# B&R Automation Studio project Panasonic_LinkaPowerCP2_A2021055 (part 11)

```iecst
			IF NOT SC_P1_StoperSrobovania.Switch1 THEN
				P1_Skrutk_5H_PravaM5_Vysunutie:= STRING_TO_REAL(Reports.Skrutkovacky.VyskaSkrutkovania.P1_PravaSkrutkaM5);
				IF (P1_Skrutk_5H_PravaM5_Vysunutie <= P1_RemPremenne.P1_Srob5H_PravaM5_Vysunutie_HI) AND (P1_Skrutk_5H_PravaM5_Vysunutie >= P1_RemPremenne.P1_Srob5H_PravaM5_Vysunutie_LO) THEN
					VysunutieSkrutkovacky_OK:= TRUE;
				ELSE
					VysunutieSkrutkovacky_OK:= FALSE;
				END_IF
				SC_P1_StoperSrobovania.Switch1:= TRUE;
			END_IF

			IF P1_Srobovanie.STAV.Vysledok_Srobovania = 'OK' THEN
				IF VysunutieSkrutkovacky_OK THEN
					Reports.Skrutkovacky.VyslednyReport.P1_PravaSkrutkaM5:= 'PASS';
					SC_P1_StoperSrobovania.ResetStep:= TRUE;
					SC_P1_StoperSrobovania.Step:= 390;
				ELSE
					Reports.Skrutkovacky.VyslednyReport.P1_PravaSkrutkaM5:= 'FAIL';
					IF P1_Srobov_M5_Result_OFF THEN
						SC_P1_StoperSrobovania.ResetStep:= TRUE;
						SC_P1_StoperSrobovania.Step:= 390;
					ELSE
						Paletka[i].PAR.StavPowerCP:= 'FAIL';
						Paletka[i].STAV.StavPaletky:= 'NG';
						SC_P1_StoperSrobovania.ResetStep:= TRUE;
						SC_P1_StoperSrobovania.Step:= 500;
					END_IF
				END_IF
			ELSIF P1_Srobovanie.STAV.Vysledok_Srobovania = 'NG' THEN
				Reports.Skrutkovacky.VyslednyReport.P1_PravaSkrutkaM5:= 'FAIL';
				IF P1_Srobov_M5_Result_OFF THEN
					SC_P1_StoperSrobovania.ResetStep:= TRUE;
					SC_P1_StoperSrobovania.Step:= 390;
				ELSE
					Paletka[i].PAR.StavPowerCP:= 'FAIL';
					Paletka[i].STAV.StavPaletky:= 'NG';
					SC_P1_StoperSrobovania.ResetStep:= TRUE;
					SC_P1_StoperSrobovania.Step:= 500;
				END_IF
			END_IF

		390:
			SC_P1_StoperSrobovania.StepName:='390 - Automaticky Rezim - model 5H odobratie skrutky M5';
			SC_P1_StoperSrobovania.IdleTime.PT:= T#200ms;
			SC_P1_StoperSrobovania.AlarmTime.PT:= T#5s;

			IF NOT SC_P1_StoperSrobovania.Switch1  THEN
				P1_Srobovanie.COM_IN.OdoberSkrutku_M5:= TRUE;
				SC_P1_StoperSrobovania.Switch1:= TRUE;
			END_IF

			IF P1_Srobovanie.STAV.ManipulatorNadPodavacmi THEN
				P1_Srobovanie.COM_IN.OdoberSkrutku_M5:= FALSE;
				SC_P1_StoperSrobovania.ResetStep:= TRUE;
				SC_P1_StoperSrobovania.Step:= 391;
			END_IF

		391:
			SC_P1_StoperSrobovania.StepName:='391 - Automaticky Rezim - cakam na zrusenie signalu presun manipulatora ukonceny';
			SC_P1_StoperSrobovania.IdleTime.PT:= T#200ms;
			SC_P1_StoperSrobovania.AlarmTime.PT:= T#5s;

			IF NOT P1_Robot.COM_IN.Stav_RobotPoziciaCakania THEN
				SC_P1_StoperSrobovania.ResetStep:= TRUE;
				SC_P1_StoperSrobovania.Step:= 392;
			END_IF

		392:
			SC_P1_StoperSrobovania.StepName:='392 - Automaticky Rezim - model 5H vystavenie signalu pre robota chod do cakacej pozicie';
			SC_P1_StoperSrobovania.IdleTime.PT:= T#200ms;
			SC_P1_StoperSrobovania.AlarmTime.PT:= T#5s;

			P1_Robot.COM_OUT.ManipSrobovania_BezpecnaPozicia:= TRUE;

			IF NOT SC_P1_StoperSrobovania.Switch1 THEN
				P1_Robot.COM_OUT.Presun_CakaciaPozicia:= TRUE;
				SC_P1_StoperSrobovania.Switch1:= TRUE;
			END_IF

			IF P1_Robot.COM_IN.Stav_RobotPoziciaCakania AND NOT P1_Srobovanie.COM_OUT.Stav_SkrutkovanieUkoncene THEN
				P1_Robot.COM_OUT.Presun_CakaciaPozicia:= FALSE;
				CAM6.STAV.Results_READY:= FALSE;
				CAM6.STAV.OldRunCounter:= CAM6.STAV.RunCounter;
				SC_P1_StoperSrobovania.ResetStep:= TRUE;
				SC_P1_StoperSrobovania.Step:= 395;
			END_IF

		395:
			SC_P1_StoperSrobovania.StepName:='395 - Inicializacia - model 5H kamerova kontrola paletky CAM6';//CAM 6//
			SC_P1_StoperSrobovania.IdleTime.PT:= T#5s;
			SC_P1_StoperSrobovania.AlarmTime.PT:= T#5s;

			IF NOT SC_P1_StoperSrobovania.Switch1 AND CAM6.STAV.Command_READY THEN
				CAM6.CMD.Triger:= TRUE;
				SC_P1_StoperSrobovania.IdleTime.IN:= TRUE;
				SC_P1_StoperSrobovania.Switch1:= TRUE;
			END_IF

			IF CAM6.STAV.Results_READY AND CAM6.STAV.Command_AKCEPTOVANY AND CAM6.STAV.OldRunCounter <> CAM6.STAV.RunCounter THEN
				PocetTrigrovKamery:= 0;
				CAM6.STAV.Results_READY:= FALSE;
				CAM6.STAV.OldRunCounter:= CAM6.STAV.RunCounter;
				SC_P1_StoperSrobovania.ResetStep:= TRUE;
				SC_P1_StoperSrobovania.Step:= 398;
			ELSIF SC_P1_StoperSrobovania.IdleTime.Q AND PocetTrigrovKamery < 5 THEN
				PocetTrigrovKamery:= PocetTrigrovKamery + 1;
				CAM6.STAV.Results_READY:= FALSE;
				CAM6.STAV.OldRunCounter:= CAM6.STAV.RunCounter;
				CAM6.CMD.Triger:= FALSE;
				SC_P1_StoperSrobovania.ResetStep:= TRUE;
				SC_P1_StoperSrobovania.Step:= 397;
			ELSIF SC_P1_StoperSrobovania.IdleTime.Q AND PocetTrigrovKamery >= 5 THEN
				P1_Alarmy[168]:= TRUE;
				P1_Pracovisko.STAV.Porucha_ST2:= TRUE;
			END_IF

		397:
			SC_P1_StoperSrobovania.StepName:='397 - Automaticky Rezim - cakam na opatovny triger kamery CAM6';
			SC_P1_StoperSrobovania.IdleTime.PT:= T#1s;
			SC_P1_StoperSrobovania.AlarmTime.PT:= T#5s;

			SC_P1_StoperSrobovania.IdleTime.IN:= TRUE;

			IF SC_P1_StoperSrobovania.IdleTime.Q THEN
				SC_P1_StoperSrobovania.ResetStep:= TRUE;
				SC_P1_StoperSrobovania.Step:= 395;
			END_IF

		398:
			SC_P1_StoperSrobovania.StepName:='398 - Automaticky Rezim - model 5H kontrola vysledku kamery';
			SC_P1_StoperSrobovania.IdleTime.PT:= T#200ms;
			SC_P1_StoperSrobovania.AlarmTime.PT:= T#5s;
			SC_P1_StoperSrobovania.IdleTime.IN:= TRUE;

			IF Linka.P1_Kamery_OFF THEN
				CAM6.CMD.Triger:= FALSE;
				CAM6.PAR.ResultFotky:= 'PASS';
				SC_P1_StoperSrobovania.ResetStep:= TRUE;
				SC_P1_StoperSrobovania.Step:= 403;
			ELSIF NOT CAM6.STAV.BUSY THEN
				CAM6.CMD.Triger:= FALSE;
				IF NOT CAM6.RESULT.Paletka.Pritom_SpodnychBusbarov_5H AND
					CAM6.RESULT.PowerCP.Pritom_LavejSkrutkyK30 AND
					CAM6.RESULT.PowerCP.Pritom_PravejSkrutkyK30 THEN
					CAM6.PAR.ResultFotky:= 'PASS';
					SC_P1_StoperSrobovania.ResetStep:= TRUE;
					SC_P1_StoperSrobovania.Step:= 403;
				ELSE
					CAM6.PAR.ResultFotky:= 'FAIL';
					SC_P1_StoperSrobovania.ResetStep:= TRUE;
					SC_P1_StoperSrobovania.Step:= 403;
				END_IF
			END_IF

		403:
			SC_P1_StoperSrobovania.StepName:='403 - Automaticky Rezim - model 5H rozhodnutie podla kamerovej kontroly paletky';
			SC_P1_StoperSrobovania.IdleTime.PT:= T#200ms;
			SC_P1_StoperSrobovania.AlarmTime.PT:= T#5s;

			IF CAM6.PAR.ResultFotky = 'PASS' THEN
				Paletka[i].PAR.StavPowerCP:= 'PASS';
				SC_P1_StoperSrobovania.ResetStep:= TRUE;
				SC_P1_StoperSrobovania.Step:= 540;
			ELSIF CAM6.PAR.ResultFotky = 'FAIL' THEN
				P1_Vizu.ZobrazHL8_ST2:= TRUE;
				IF P1_Srobov_KAM_Result_OK THEN
					P1_Srobov_KAM_Result_OK:= FALSE;
					P1_Vizu.ZobrazHL8_ST2:= FALSE;
					Paletka[i].PAR.StavPowerCP:= 'PASS';
					CAM6.PAR.ResultFotky:= 'PASS';
					SC_P1_StoperSrobovania.ResetStep:= TRUE;
					SC_P1_StoperSrobovania.Step:= 540;
				ELSIF P1_Srobov_KAM_Result_NG THEN
					P1_Srobov_KAM_Result_NG:= FALSE;
					P1_Vizu.ZobrazHL8_ST2:= FALSE;
					Paletka[i].PAR.StavPowerCP:= 'FAIL';
					Paletka[i].STAV.StavPaletky:= 'NG';
					SC_P1_StoperSrobovania.ResetStep:= TRUE;
					SC_P1_StoperSrobovania.Step:= 540;
				END_IF
			END_IF

			//**************************Uvolnenie robota a vyfotenie paletky po zlom skrutkovaní*****************************************************//

		500:
			SC_P1_StoperSrobovania.StepName:='500 - Automaticky Rezim - presun manipulatora vzad';
			SC_P1_StoperSrobovania.IdleTime.PT:= T#200ms;
			SC_P1_StoperSrobovania.AlarmTime.PT:= T#5s;

			IF NOT SC_P1_StoperSrobovania.Switch1 THEN
				P1_Srobovanie.COM_IN.PresunManipulatora_VZAD:= TRUE;
				SC_P1_StoperSrobovania.Switch1:= TRUE;
			END_IF

			IF P1_Srobovanie.COM_OUT.Stav_PresunManipulUkonceny THEN
				P1_Srobovanie.COM_IN.PresunManipulatora_VZAD:= FALSE;
				SC_P1_StoperSrobovania.ResetStep:= TRUE;
				SC_P1_StoperSrobovania.Step:= 501;
			END_IF

		501:
			SC_P1_StoperSrobovania.StepName:='501 - Automaticky Rezim - cakam na zrusenie signalu presun manipulatora ukonceny';
			SC_P1_StoperSrobovania.IdleTime.PT:= T#200ms;
			SC_P1_StoperSrobovania.AlarmTime.PT:= T#5s;

			IF NOT P1_Srobovanie.COM_OUT.Stav_PresunManipulUkonceny THEN
				SC_P1_StoperSrobovania.ResetStep:= TRUE;
				SC_P1_StoperSrobovania.Step:= 503;
			END_IF

		503:
			SC_P1_StoperSrobovania.StepName:='503 - Automaticky Rezim - kontrola ci robot drzi foamy';
			SC_P1_StoperSrobovania.IdleTime.PT:= T#200ms;
			SC_P1_StoperSrobovania.AlarmTime.PT:= T#5s;

			IF Linka.PAR.ZvolenyModel = '4F' THEN
				IF P1_Robot.STAV.DrziFoamy_45F THEN
					P1_Robot.COM_OUT.PolozFoam4F_na_PowerCP:= TRUE;
					IF P1_Robot.COM_IN.Stav_Foam4F_Polozeny THEN
						P1_Robot.COM_OUT.PolozFoam4F_na_PowerCP:= FALSE;
						SC_P1_StoperSrobovania.ResetStep:= TRUE;
						SC_P1_StoperSrobovania.Step:= 505;
					END_IF
				ELSE
					SC_P1_StoperSrobovania.ResetStep:= TRUE;
					SC_P1_StoperSrobovania.Step:= 505;
				END_IF
			ELSIF Linka.PAR.ZvolenyModel = '5F' THEN
				IF P1_Robot.STAV.DrziFoamy_45F THEN
					P1_Robot.COM_OUT.PolozFoam5F_na_PowerCP:= TRUE;
					IF P1_Robot.COM_IN.Stav_Foam5F_Polozeny THEN
						P1_Robot.COM_OUT.PolozFoam5F_na_PowerCP:= FALSE;
						SC_P1_StoperSrobovania.ResetStep:= TRUE;
						SC_P1_StoperSrobovania.Step:= 505;
					END_IF
				ELSE
					SC_P1_StoperSrobovania.ResetStep:= TRUE;
					SC_P1_StoperSrobovania.Step:= 505;
				END_IF
			ELSIF Linka.PAR.ZvolenyModel = '5H' THEN
				SC_P1_StoperSrobovania.ResetStep:= TRUE;
				SC_P1_StoperSrobovania.Step:= 505;
			END_IF

		505:
			SC_P1_StoperSrobovania.StepName:='505 - Automaticky Rezim - kontrola ci robot drzi busbary';
			SC_P1_StoperSrobovania.IdleTime.PT:= T#200ms;
			SC_P1_StoperSrobovania.AlarmTime.PT:= T#5s;

			IF Linka.PAR.ZvolenyModel = '4F' THEN
				IF P1_Robot.STAV.DrziBusbar_45F THEN
					P1_Robot.COM_OUT.PolozSpodnyBusbar4F_na_PowerCP:= TRUE;
					IF P1_Robot.COM_IN.Stav_SpodnyBusbar4F_Polozeny THEN
						P1_Robot.COM_OUT.PolozSpodnyBusbar4F_na_PowerCP:= FALSE;
						SC_P1_StoperSrobovania.ResetStep:= TRUE;
						SC_P1_StoperSrobovania.Step:= 508;
					END_IF
				ELSE
					SC_P1_StoperSrobovania.ResetStep:= TRUE;
					SC_P1_StoperSrobovania.Step:= 508;
				END_IF
			ELSIF Linka.PAR.ZvolenyModel = '5F' THEN
				IF P1_Robot.STAV.DrziBusbar_45F THEN
					P1_Robot.COM_OUT.PolozSpodnyBusbar5F_na_PowerCP:= TRUE;
					IF P1_Robot.COM_IN.Stav_SpodnyBusbar5F_Polozeny THEN
						P1_Robot.COM_OUT.PolozSpodnyBusbar5F_na_PowerCP:= FALSE;
						SC_P1_StoperSrobovania.ResetStep:= TRUE;
						SC_P1_StoperSrobovania.Step:= 508;
					END_IF
				ELSE
					SC_P1_StoperSrobovania.ResetStep:= TRUE;
					SC_P1_StoperSrobovania.Step:= 508;
				END_IF
			ELSIF Linka.PAR.ZvolenyModel = '5H' THEN
				IF P1_Robot.STAV.DrziBusbar_5H THEN
					P1_Robot.COM_OUT.PolozSpodnyBusbar5H_na_PowerCP:= TRUE;
					IF P1_Robot.COM_IN.Stav_SpodnyBusbar5H_Polozeny THEN
						P1_Robot.COM_OUT.PolozSpodnyBusbar5H_na_PowerCP:= FALSE;
						SC_P1_StoperSrobovania.ResetStep:= TRUE;
						SC_P1_StoperSrobovania.Step:= 510;
					END_IF
				ELSE
					SC_P1_StoperSrobovania.ResetStep:= TRUE;
					SC_P1_StoperSrobovania.Step:= 510;
				END_IF
			END_IF

		508:
			SC_P1_StoperSrobovania.StepName:='508 - Automaticky Rezim - kontrola ci robot drzi DPS';
			SC_P1_StoperSrobovania.IdleTime.PT:= T#200ms;
			SC_P1_StoperSrobovania.AlarmTime.PT:= T#5s;

			IF Linka.PAR.ZvolenyModel = '4F' THEN
				IF P1_Robot.STAV.DrziDPS_45F THEN
					P1_Robot.COM_OUT.PolozDPS_4F_na_PowerCP:= TRUE;
					IF P1_Robot.COM_IN.Stav_DPS_4F_Polozeny THEN
						P1_Robot.COM_OUT.PolozDPS_4F_na_PowerCP:= FALSE;
						SC_P1_StoperSrobovania.ResetStep:= TRUE;
						SC_P1_StoperSrobovania.Step:= 510;
					END_IF
				ELSE
					SC_P1_StoperSrobovania.ResetStep:= TRUE;
					SC_P1_StoperSrobovania.Step:= 510;
				END_IF
			ELSIF Linka.PAR.ZvolenyModel = '5F' THEN
				IF P1_Robot.STAV.DrziDPS_45F THEN
					P1_Robot.COM_OUT.PolozDPS_5F_na_PowerCP:= TRUE;
					IF P1_Robot.COM_IN.Stav_DPS_5F_Polozeny THEN
						P1_Robot.COM_OUT.PolozDPS_5F_na_PowerCP:= FALSE;
						SC_P1_StoperSrobovania.ResetStep:= TRUE;
						SC_P1_StoperSrobovania.Step:= 510;
					END_IF
				ELSE
					SC_P1_StoperSrobovania.ResetStep:= TRUE;
					SC_P1_StoperSrobovania.Step:= 510;
				END_IF
			END_IF

		510:
			SC_P1_StoperSrobovania.StepName:='510 - Automaticky Rezim - vystavenie signalu pre robota chod do cakacej pozicie';
			SC_P1_StoperSrobovania.IdleTime.PT:= T#200ms;
			SC_P1_StoperSrobovania.AlarmTime.PT:= T#5s;

			P1_Robot.COM_OUT.ManipSrobovania_BezpecnaPozicia:= TRUE;

			IF NOT SC_P1_StoperSrobovania.Switch1 THEN
				P1_Robot.COM_OUT.Presun_CakaciaPozicia:= TRUE;
				SC_P1_StoperSrobovania.Switch1:= TRUE;
			END_IF

			IF P1_Robot.COM_IN.Stav_RobotPoziciaCakania THEN
				P1_Robot.COM_OUT.Presun_CakaciaPozicia:= FALSE;
				CAM6.STAV.Results_READY:= FALSE;
				CAM6.STAV.OldRunCounter:= CAM6.STAV.RunCounter;
				SC_P1_StoperSrobovania.ResetStep:= TRUE;
				SC_P1_StoperSrobovania.Step:= 513;
			END_IF

		513:
			SC_P1_StoperSrobovania.StepName:='513 - Automaticky Rezim - kamerova kontrola paletky CAM6';//CAM 6//
			SC_P1_StoperSrobovania.IdleTime.PT:= T#5s;
			SC_P1_StoperSrobovania.AlarmTime.PT:= T#5s;

			IF NOT SC_P1_StoperSrobovania.Switch1 AND CAM6.STAV.Command_READY THEN
				CAM6.CMD.Triger:= TRUE;
				SC_P1_StoperSrobovania.IdleTime.IN:= TRUE;
				SC_P1_StoperSrobovania.Switch1:= TRUE;
			END_IF

			IF CAM6.STAV.Results_READY AND CAM6.STAV.Command_AKCEPTOVANY AND CAM6.STAV.OldRunCounter <> CAM6.STAV.RunCounter THEN
				PocetTrigrovKamery:= 0;
				CAM6.STAV.Results_READY:= FALSE;
				CAM6.STAV.OldRunCounter:= CAM6.STAV.RunCounter;
				CAM6.PAR.ResultFotky:= 'FAIL';
				CAM6.CMD.Triger:= FALSE;
				SC_P1_StoperSrobovania.ResetStep:= TRUE;
				SC_P1_StoperSrobovania.Step:= 540;
			ELSIF SC_P1_StoperSrobovania.IdleTime.Q AND PocetTrigrovKamery < 5 THEN
				PocetTrigrovKamery:= PocetTrigrovKamery + 1;
				CAM6.STAV.Results_READY:= FALSE;
				CAM6.STAV.OldRunCounter:= CAM6.STAV.RunCounter;
				CAM6.CMD.Triger:= FALSE;
				SC_P1_StoperSrobovania.ResetStep:= TRUE;
				SC_P1_StoperSrobovania.Step:= 515;
			ELSIF SC_P1_StoperSrobovania.IdleTime.Q AND PocetTrigrovKamery >= 5 THEN
				P1_Alarmy[168]:= TRUE;
				P1_Pracovisko.STAV.Porucha_ST2:= TRUE;
			END_IF

		515:
			SC_P1_StoperSrobovania.StepName:='506 - Automaticky Rezim - cakam na opatovny triger kamery CAM6';
			SC_P1_StoperSrobovania.IdleTime.PT:= T#1s;
			SC_P1_StoperSrobovania.AlarmTime.PT:= T#5s;
			SC_P1_StoperSrobovania.IdleTime.IN:= TRUE;

			IF SC_P1_StoperSrobovania.IdleTime.Q THEN
				SC_P1_StoperSrobovania.ResetStep:= TRUE;
				SC_P1_StoperSrobovania.Step:= 513;
			END_IF

			//**************************Odoslanie fotiek na server************************************//

		540:
			SC_P1_StoperSrobovania.StepName:='540 - Automaticky Rezim - odoslanie fotiek na server Panasonic';
			SC_P1_StoperSrobovania.IdleTime.PT:= T#200ms;
			SC_P1_StoperSrobovania.AlarmTime.PT:= T#5s;

			IF Linka.KOM_FTP_OFF THEN
				SC_P1_StoperSrobovania.ResetStep:= TRUE;
				SC_P1_StoperSrobovania.Step:= 545;
			ELSIF NOT SC_P1_StoperSrobovania.Switch1 THEN
				FTP_CAM6.INPUTS.QRkodPowerCP:= Paletka[i].PAR.QRkodPowerCP;
				CisloFotky:= CisloFotky + 1;
				FTP_CAM6.INPUTS.IndexFotky:= USINT_TO_STRING(CisloFotky);
				FTP_CAM6.INPUTS.Result:= CAM6.PAR.ResultFotky;
				Reports.Kamery.P1_CAM6_KontrolaPaletky:= CAM6.PAR.ResultFotky;
				FTP_CAM6.CMD.OdosliFotku:= TRUE;
				P1_Skrutkovanie_Taktime.IN.START_MeraniaStratovehoCasu:= TRUE;
				SC_P1_StoperSrobovania.Switch1:= TRUE;
			END_IF

			IF FTP_CAM6.STATUS.KomunikaciaUkoncena THEN
				FTP_CAM6.CMD.OdosliFotku:= FALSE;
				P1_Skrutkovanie_Taktime.IN.START_MeraniaStratovehoCasu:= FALSE;
				Paletka[i].STAV.OdoslanieFotiek_DONE:= TRUE;
				SC_P1_StoperSrobovania.ResetStep:= TRUE;
				SC_P1_StoperSrobovania.Step:= 545;
			ELSIF FTP_CAM6.STATUS.KomunikaciaError THEN
				P1_Skrutkovanie_Taktime.IN.START_MeraniaStratovehoCasu:= FALSE;
				P1_Alarmy[116]:= TRUE;
				P1_Pracovisko.STAV.Porucha_ST2:= TRUE;
			END_IF

			//******************Odcentrovanie paletky************************************//
		545:
			SC_P1_StoperSrobovania.StepName:='545 - Automaticky Rezim - odcentrovanie paletky';
			SC_P1_StoperSrobovania.IdleTime.PT:= T#200ms;
			SC_P1_StoperSrobovania.AlarmTime.PT:= T#5s;

			IF NOT SC_P1_StoperSrobovania.Switch1 THEN
				Centrovacku_ZASUN:= TRUE;
				SC_P1_StoperSrobovania.Switch1:= TRUE;
			END_IF

			IF P1_StoperSrobovania.IN.Centrovanie_ZASUNUTE THEN
				P1_Srobovanie.COM_IN.OdoberSkrutku_M5:= FALSE;
				SC_P1_StoperSrobovania.ResetStep:= TRUE;
				SC_P1_StoperSrobovania.Step:= 548;
			END_IF

		548:
			SC_P1_StoperSrobovania.StepName:='548 - Automaticky Rezim - cakam na zrusenie signalu skrutkovanie ukoncene';
			SC_P1_StoperSrobovania.IdleTime.PT:= T#200ms;
			SC_P1_StoperSrobovania.AlarmTime.PT:= T#5s;

			IF NOT P1_Srobovanie.COM_OUT.Stav_SkrutkovanieUkoncene THEN
				SC_P1_StoperSrobovania.ResetStep:= TRUE;
				SC_P1_StoperSrobovania.Step:= 550;
			END_IF

			//**************************Odoslanie dát na server******************************************//

		550:
			SC_P1_StoperSrobovania.StepName:='550 - Automaticky Rezim - odoslanie stavu paletky na server';
			SC_P1_StoperSrobovania.IdleTime.PT:= T#200ms;
			SC_P1_StoperSrobovania.AlarmTime.PT:= T#10s;

			IF Linka.KOM_Panatrace_OFF THEN
				SC_P1_StoperSrobovania.ResetStep:= TRUE;
				SC_P1_StoperSrobovania.Step:= 560;
			ELSIF NOT SC_P1_StoperSrobovania.Switch1 AND TRCB_P1_Srobovanie_ST2.STATUS.KOM_READY THEN
				TRCB_P1_Srobovanie_ST2.CMD.OdosliStavPaletky_TYP2:= TRUE;
				(*P1_Skrutkovanie_Taktime.IN.START_MeraniaStratovehoCasu:= TRUE;*)
				SC_P1_StoperSrobovania.Switch1:= TRUE;
			END_IF

			IF TRCB_P1_Srobovanie_ST2.STATUS.KomunikaciaUkoncena THEN
				TRCB_P1_Srobovanie_ST2.CMD.OdosliStavPaletky_TYP2:= FALSE;
				P1_Skrutkovanie_Taktime.IN.START_MeraniaStratovehoCasu:= FALSE;
				SC_P1_StoperSrobovania.ResetStep:= TRUE;
				SC_P1_StoperSrobovania.Step:= 552;
			ELSIF TRCB_P1_Srobovanie_ST2.STATUS.KomunikaciaError THEN
				TRCB_P1_Srobovanie_ST2.CMD.OdosliStavPaletky_TYP2:= FALSE;
				P1_Skrutkovanie_Taktime.IN.START_MeraniaStratovehoCasu:= FALSE;
				SC_P1_StoperSrobovania.ResetStep:= TRUE;
				SC_P1_StoperSrobovania.Step:= 557;
			END_IF

		552:
			SC_P1_StoperSrobovania.StepName:='552 - Automaticky Rezim - kontrola odpovede servera';
			SC_P1_StoperSrobovania.IdleTime.PT:= T#200ms;
			SC_P1_StoperSrobovania.AlarmTime.PT:= T#10s;

			IF NOT TRCB_P1_Srobovanie_ST2.STATUS.KomunikaciaUkoncena THEN
				IF TRCB_P1_Srobovanie_ST2.OUTPUTS.PovolenieCinnostiNaPaletke = 'OK' THEN
					Paletka[i].STAV.Komunikacia_DONE:= TRUE;
					P1_StoperSrobovania.STAV.VyrobaZacala:= FALSE;
					SC_P1_StoperSrobovania.ResetStep:= TRUE;
					SC_P1_StoperSrobovania.Step:= 560;
				ELSIF TRCB_P1_Srobovanie_ST2.OUTPUTS.PovolenieCinnostiNaPaletke = 'NG' THEN
					Paletka[i].STAV.StavPaletky:= 'NG';
					P1_StoperSrobovania.STAV.VyrobaZacala:= FALSE;
					SC_P1_StoperSrobovania.ResetStep:= TRUE;
					SC_P1_StoperSrobovania.Step:= 560;
				END_IF
			END_IF

		555:
			SC_P1_StoperSrobovania.StepName:='555 - Automaticky Rezim - vyziadanie stavu komunikacie zo serverom';
			SC_P1_StoperSrobovania.IdleTime.PT:= T#200ms;
			SC_P1_StoperSrobovania.AlarmTime.PT:= T#10s;

			IF NOT SC_P1_StoperSrobovania.Switch1 AND TRCB_P1_Srobovanie_ST2.STATUS.KOM_READY THEN
				TRCB_P1_Srobovanie_ST2.CMD.VyziadajStavPanatrace_TYP4:= TRUE;
				SC_P1_StoperSrobovania.Switch1:= TRUE;
			END_IF

			IF TRCB_P1_Srobovanie_ST2.STATUS.KomunikaciaUkoncena THEN
				TRCB_P1_Srobovanie_ST2.CMD.VyziadajStavPanatrace_TYP4:= FALSE;
				SC_P1_StoperSrobovania.ResetStep:= TRUE;
				SC_P1_StoperSrobovania.Step:= 556;
			ELSIF TRCB_P1_Srobovanie_ST2.STATUS.KomunikaciaError THEN
				TRCB_P1_Srobovanie_ST2.CMD.VyziadajStavPanatrace_TYP4:= FALSE;
				SC_P1_StoperSrobovania.ResetStep:= TRUE;
				SC_P1_StoperSrobovania.Step:= 557;
			END_IF

		556:
			SC_P1_StoperSrobovania.StepName:='556 - Automaticky Rezim - kontrola odpovede servera';
			SC_P1_StoperSrobovania.IdleTime.PT:= T#200ms;
			SC_P1_StoperSrobovania.AlarmTime.PT:= T#5s;

			IF NOT TRCB_P1_Srobovanie_ST2.STATUS.KomunikaciaUkoncena THEN
				IF TRCB_P1_Srobovanie_ST2.OUTPUTS.DruhCinnostiNaPaletke = '0;Generating' THEN
					SC_P1_StoperSrobovania.ResetStep:= TRUE;
					SC_P1_StoperSrobovania.Step:= 557;
				ELSIF TRCB_P1_Srobovanie_ST2.OUTPUTS.DruhCinnostiNaPaletke = '1;Request' THEN
					SC_P1_StoperSrobovania.ResetStep:= TRUE;
					SC_P1_StoperSrobovania.Step:= 557;
				ELSIF TRCB_P1_Srobovanie_ST2.OUTPUTS.DruhCinnostiNaPaletke = '2;Report' THEN
					SC_P1_StoperSrobovania.ResetStep:= TRUE;
					SC_P1_StoperSrobovania.Step:= 550;
				ELSIF TRCB_P1_Srobovanie_ST2.OUTPUTS.DruhCinnostiNaPaletke = '3;Wedding' THEN
					SC_P1_StoperSrobovania.ResetStep:= TRUE;
					SC_P1_StoperSrobovania.Step:= 557;
				ELSIF TRCB_P1_Srobovanie_ST2.OUTPUTS.DruhCinnostiNaPaletke = '4;Status' THEN
					SC_P1_StoperSrobovania.ResetStep:= TRUE;
					SC_P1_StoperSrobovania.Step:= 557;
				ELSIF TRCB_P1_Srobovanie_ST2.OUTPUTS.DruhCinnostiNaPaletke = '5;' THEN
					SC_P1_StoperSrobovania.ResetStep:= TRUE;
					SC_P1_StoperSrobovania.Step:= 557;
				ELSE
					SC_P1_StoperSrobovania.ResetStep:= TRUE;
					SC_P1_StoperSrobovania.Step:= 557;
				END_IF
			END_IF

		557:
			SC_P1_StoperSrobovania.StepName:='557 - Automaticky Rezim - rozhodnutie obsluhy po chybe komunikacie s Panatrace';
			SC_P1_StoperSrobovania.IdleTime.PT:= T#200ms;
			SC_P1_StoperSrobovania.AlarmTime.PT:= T#5s;

			P1_Vizu.ZobrazHL10_ST2:= TRUE;

			IF TRCB_P1_Srobov_OpatovnyDopyt THEN
				TRCB_P1_Srobov_OpatovnyDopyt:= FALSE;
				P1_Vizu.ZobrazHL10_ST2:= FALSE;
				SC_P1_StoperSrobovania.ResetStep:= TRUE;
				SC_P1_StoperSrobovania.Step:= 555;
			ELSIF TRCB_P1_Srobov_PaletkaNG THEN
				TRCB_P1_Srobov_PaletkaNG:= FALSE;
				P1_Vizu.ZobrazHL10_ST2:= FALSE;
				Paletka[i].STAV.StavPaletky := 'NG';
				P1_StoperSrobovania.STAV.VyrobaZacala:= FALSE;
				SC_P1_StoperSrobovania.ResetStep:= TRUE;
				SC_P1_StoperSrobovania.Step:= 560;
			END_IF

			//***********************************Vyvezenie paletky**************************************************//

		560:
			SC_P1_StoperSrobovania.StepName:='560 - Automaticky Rezim - cakam na vyvezenie na akumulacny stoper';
			SC_P1_StoperSrobovania.IdleTime.PT:= T#200ms;
			SC_P1_StoperSrobovania.AlarmTime.PT:= T#5s;

			IF P1_StoperSrobovania.KoniecCyklu THEN
				SC_P1_StoperSrobovania.ResetStep:= TRUE;
				SC_P1_StoperSrobovania.Step:= 0;
			ELSIF P1_Pracovisko.STAV.Porucha_ST2 THEN
				SC_P1_StoperSrobovania.ResetStep:= TRUE;
				SC_P1_StoperSrobovania.Step:= 0;
			ELSIF NOT P1_AkumulacnyStoper.IN.PritomnostPaletky AND SC_P1_AkumulacnyStoper.Step = 100 AND NOT P1_StoperSrobovania.STAV.PrebiehaVyvezeniePaletky AND Safety.STAV.P1_VystupBunky_VystupBar_AKTIVNA THEN
				P1_StoperSrobovania.OUT.ZasunStoper:= TRUE;
				P1_StoperSrobovania.STAV.PrebiehaVyvezeniePaletky:= TRUE;
				SC_P1_StoperSrobovania.ResetStep:= TRUE;
				SC_P1_StoperSrobovania.Step:= 561;
			END_IF

		561:
			SC_P1_StoperSrobovania.StepName:='561 - Automaticky Rezim - ukoncenie vyvazania na akumulacny stoper';
			SC_P1_StoperSrobovania.IdleTime.PT:= T#200ms;
			SC_P1_StoperSrobovania.AlarmTime.PT:= T#10s;

			SC_P1_StoperSrobovania.AlarmTime.IN:= P1_StoperSrobovania.RFID_hlava.PritomnostPaletky;
			SC_P1_StoperSrobovania.IdleTime.IN:= NOT P1_StoperSrobovania.RFID_hlava.PritomnostPaletky;

			IF NOT P1_StoperSrobovania.RFID_hlava.PritomnostPaletky THEN
				TestovaciKus:= FALSE;
				CisloFotky:= 0;
				Paletka[i].PAR.StavPowerCP:= '';
				Paletka[i].STAV.Komunikacia_DONE:= FALSE;
				Paletka[i].STAV.OdoslanieFotiek_DONE:= FALSE;
				Reports.Skrutkovacky.Moment_ToleranciaMIN.P1_LavaSkrutkaK30:= '';
				Reports.Skrutkovacky.Moment_ToleranciaMAX.P1_LavaSkrutkaK30:= '';
				Reports.Skrutkovacky.Moment_NameranaHodnota.P1_LavaSkrutkaK30:= '';
				Reports.Skrutkovacky.VyslednyReport.P1_LavaSkrutkaK30:= '';
				Reports.Skrutkovacky.Uhol_ToleranciaMIN.P1_LavaSkrutkaK30:= '';
				Reports.Skrutkovacky.Uhol_ToleranciaMAX.P1_LavaSkrutkaK30:= '';
				Reports.Skrutkovacky.Uhol_NameranaHodnota.P1_LavaSkrutkaK30:= '';
				Reports.Skrutkovacky.CasSkrutkovania.P1_LavaSkrutkaK30:= '';
				Reports.Skrutkovacky.VyslednyReport.P1_LavaSkrutkaK30:= '';
				Reports.Skrutkovacky.VyskaSkrutkovania.P1_LavaSkrutkaK30:= '';
				Reports.Skrutkovacky.Moment_ToleranciaMIN.P1_PravaSkrutkaK30:= '';
				Reports.Skrutkovacky.Moment_ToleranciaMAX.P1_PravaSkrutkaK30:= '';
				Reports.Skrutkovacky.Moment_NameranaHodnota.P1_PravaSkrutkaK30:= '';
				Reports.Skrutkovacky.VyslednyReport.P1_PravaSkrutkaK30:= '';
				Reports.Skrutkovacky.Uhol_ToleranciaMIN.P1_PravaSkrutkaK30:= '';
				Reports.Skrutkovacky.Uhol_ToleranciaMAX.P1_PravaSkrutkaK30:= '';
				Reports.Skrutkovacky.Uhol_NameranaHodnota.P1_PravaSkrutkaK30:= '';
				Reports.Skrutkovacky.CasSkrutkovania.P1_PravaSkrutkaK30:= '';
				Reports.Skrutkovacky.VyskaSkrutkovania.P1_PravaSkrutkaK30:= '';
				Reports.Skrutkovacky.Moment_ToleranciaMIN.P1_ZadnaSkrutkaM4:= '';
				Reports.Skrutkovacky.Moment_ToleranciaMAX.P1_ZadnaSkrutkaM4:= '';
				Reports.Skrutkovacky.Moment_NameranaHodnota.P1_ZadnaSkrutkaM4:= '';
				Reports.Skrutkovacky.VyslednyReport.P1_ZadnaSkrutkaM4:= '';
				Reports.Skrutkovacky.Uhol_ToleranciaMIN.P1_ZadnaSkrutkaM4:= '';
				Reports.Skrutkovacky.Uhol_ToleranciaMAX.P1_ZadnaSkrutkaM4:= '';
				Reports.Skrutkovacky.Uhol_NameranaHodnota.P1_ZadnaSkrutkaM4:= '';
				Reports.Skrutkovacky.CasSkrutkovania.P1_ZadnaSkrutkaM4:= '';
				Reports.Skrutkovacky.VyskaSkrutkovania.P1_ZadnaSkrutkaM4:= '';
				Reports.Skrutkovacky.Moment_ToleranciaMIN.P1_PrednaSkrutkaM4:= '';
				Reports.Skrutkovacky.Moment_ToleranciaMAX.P1_PrednaSkrutkaM4:= '';
				Reports.Skrutkovacky.Moment_NameranaHodnota.P1_PrednaSkrutkaM4:= '';
				Reports.Skrutkovacky.VyslednyReport.P1_PrednaSkrutkaM4:= '';
				Reports.Skrutkovacky.Uhol_ToleranciaMIN.P1_PrednaSkrutkaM4:= '';
				Reports.Skrutkovacky.Uhol_ToleranciaMAX.P1_PrednaSkrutkaM4:= '';
				Reports.Skrutkovacky.Uhol_NameranaHodnota.P1_PrednaSkrutkaM4:= '';
				Reports.Skrutkovacky.CasSkrutkovania.P1_PrednaSkrutkaM4:= '';
				Reports.Skrutkovacky.VyskaSkrutkovania.P1_PrednaSkrutkaM4:= '';
				Reports.Skrutkovacky.Moment_ToleranciaMIN.P1_SkrutkaDPS_M4:= '';
				Reports.Skrutkovacky.Moment_ToleranciaMAX.P1_SkrutkaDPS_M4:= '';
				Reports.Skrutkovacky.Moment_NameranaHodnota.P1_SkrutkaDPS_M4:= '';
				Reports.Skrutkovacky.VyslednyReport.P1_SkrutkaDPS_M4:= '';
				Reports.Skrutkovacky.Uhol_ToleranciaMIN.P1_SkrutkaDPS_M4:= '';
				Reports.Skrutkovacky.Uhol_ToleranciaMAX.P1_SkrutkaDPS_M4:= '';
				Reports.Skrutkovacky.Uhol_NameranaHodnota.P1_SkrutkaDPS_M4:= '';
				Reports.Skrutkovacky.CasSkrutkovania.P1_SkrutkaDPS_M4:= '';
				Reports.Skrutkovacky.VyskaSkrutkovania.P1_SkrutkaDPS_M4:= '';
				Reports.Skrutkovacky.Moment_ToleranciaMIN.P1_LavaSkrutkaM5:= '';
				Reports.Skrutkovacky.Moment_ToleranciaMAX.P1_LavaSkrutkaM5:= '';
				Reports.Skrutkovacky.Moment_NameranaHodnota.P1_LavaSkrutkaM5:= '';
				Reports.Skrutkovacky.VyslednyReport.P1_LavaSkrutkaM5:= '';
				Reports.Skrutkovacky.Uhol_ToleranciaMIN.P1_LavaSkrutkaM5:= '';
				Reports.Skrutkovacky.Uhol_ToleranciaMAX.P1_LavaSkrutkaM5:= '';
				Reports.Skrutkovacky.Uhol_NameranaHodnota.P1_LavaSkrutkaM5:= '';
				Reports.Skrutkovacky.CasSkrutkovania.P1_LavaSkrutkaM5:= '';
				Reports.Skrutkovacky.VyskaSkrutkovania.P1_LavaSkrutkaM5:= '';
				Reports.Skrutkovacky.Moment_ToleranciaMIN.P1_PravaSkrutkaM5:= '';
				Reports.Skrutkovacky.Moment_ToleranciaMAX.P1_PravaSkrutkaM5:= '';
				Reports.Skrutkovacky.Moment_NameranaHodnota.P1_PravaSkrutkaM5:= '';
				Reports.Skrutkovacky.VyslednyReport.P1_PravaSkrutkaM5:= '';
				Reports.Skrutkovacky.Uhol_ToleranciaMIN.P1_PravaSkrutkaM5:= '';
				Reports.Skrutkovacky.Uhol_ToleranciaMAX.P1_PravaSkrutkaM5:= '';
				Reports.Skrutkovacky.Uhol_NameranaHodnota.P1_PravaSkrutkaM5:= '';
				Reports.Skrutkovacky.CasSkrutkovania.P1_PravaSkrutkaM5:= '';
				Reports.Skrutkovacky.VyskaSkrutkovania.P1_PravaSkrutkaM5:= '';
				Reports.Skrutkovacky.Moment_ToleranciaMIN.P1_StrednaSkrutkaM5:= '';
				Reports.Skrutkovacky.Moment_ToleranciaMAX.P1_StrednaSkrutkaM5:= '';
				Reports.Skrutkovacky.Moment_NameranaHodnota.P1_StrednaSkrutkaM5:= '';
				Reports.Skrutkovacky.VyslednyReport.P1_StrednaSkrutkaM5:= '';
				Reports.Skrutkovacky.Uhol_ToleranciaMIN.P1_StrednaSkrutkaM5:= '';
				Reports.Skrutkovacky.Uhol_ToleranciaMAX.P1_StrednaSkrutkaM5:= '';
				Reports.Skrutkovacky.Uhol_NameranaHodnota.P1_StrednaSkrutkaM5:= '';
				Reports.Skrutkovacky.CasSkrutkovania.P1_StrednaSkrutkaM5:= '';
				Reports.Skrutkovacky.VyskaSkrutkovania.P1_StrednaSkrutkaM5:= '';
				Reports.Kamery.P1_CAM6_KontrolaPaletky:= '';
				P1_Robot.STAV.DrziBusbar_45F:= FALSE;
				P1_Robot.STAV.DrziBusbar_5H:= FALSE;
				P1_Robot.STAV.DrziDPS_45F:= FALSE;
				P1_Robot.STAV.DrziFoamy_45F:= FALSE;
				P1_StoperSrobovania.OUT.ZasunStoper:= FALSE;
				P1_Srobovanie.COM_OUT.Stav_PoruchaSkrutkovania:= FALSE;
				P1_StoperSrobovania.STAV.VstupnaKamerovaKontrola:= FALSE;
				SC_P1_StoperSrobovania.ResetStep:= TRUE;
				SC_P1_StoperSrobovania.Step:= 100;
			ELSIF SC_P1_StoperSrobovania.AlarmTime.Q THEN
				P1_Alarmy[161]:= TRUE;
				P1_Pracovisko.STAV.Porucha_ST2:= TRUE;
			END_IF

			//*******************************************************Manuálny režim*******************************************************************************//

		700:
			SC_P1_StoperSrobovania.StepName:='700 - Manualny Rezim';
			SC_P1_StoperSrobovania.IdleTime.PT:= T#8s;
			SC_P1_StoperSrobovania.AlarmTime.PT:= T#5s;

			//Ovládanie zdvižky//
			IF P1_StoperSrobovania.CMD.RR_VysunCentrovanie THEN
				P1_StoperSrobovania.OUT.Centrovanie_ZASUN:= FALSE;
				P1_StoperSrobovania.OUT.Centrovanie_VYSUN:= TRUE;
			ELSE
				P1_StoperSrobovania.OUT.Centrovanie_ZASUN:= TRUE;
				P1_StoperSrobovania.OUT.Centrovanie_VYSUN:= FALSE;
			END_IF

	END_CASE
				END_PROGRAM

PROGRAM _EXIT
				(* Insert code here *)

				END_PROGRAM
```

#### Variables.var - Local variables
```iecst
VAR
	SC_OvlCentrovacky : SequenceControlTyp;
	Centrovacku_VYSUN : BOOL;
	Centrovacku_ZASUN : BOOL;
	i : USINT;
	VysunutieSkrutkovacky_OK : BOOL := 0;
	PocetTrigrovKamery : USINT := 0;
	PocetDopytovNaServer : USINT := 0;
	PocetZopakovaniOdobratia : USINT := 0;
	TestovaciKus : BOOL := 0;
	P1_Skrutk_45F_LavaK30_Vysunutie : REAL := 0.0;
	P1_Skrutk_45F_PravaK30_Vysunutie : REAL := 0.0;
	P1_Skrutk_45F_PrednaM4_Vysunutie : REAL := 0.0;
	P1_Skrutk_45F_ZadnaM4_Vysunutie : REAL := 0.0;
	CisloFotky : USINT := 0;
	P1_Skrutk_45F_DPS_M4_Vysunutie : REAL := 0.0;
	P1_Skrutk_5H_LavaK30_Vysunutie : REAL := 0.0;
	P1_Skrutk_5H_PravaK30_Vysunutie : REAL := 0.0;
	P1_Skrutk_5H_StrednaM5_Vysunutie : REAL := 0.0;
	P1_Skrutk_5H_LavaM5_Vysunutie : REAL := 0.0;
	P1_Skrutk_5H_PravaM5_Vysunutie : REAL := 0.0;
	Triger_0 : BOOL := 0;
	Round_0 : Round;
END_VAR
```

#### IOLinkKomunikacia.st
```iecst
ACTION IOLinkKomunikacia:

	//RFID snímač paletky//
	P1_StoperSrobovania.RFID_hlava();

	//Snímač vysunutia skrutkovačky K30//
	Round_0.VstupnaHodnota:= P1_Srobovanie.PAR.Skrutkov_K30_AktualHodnVysunutia;
	P1_Srobovanie.PAR.Skrutkov_K30_RoundHodnotaREAL:= Round_0.VystupnaHodnota;
	Round_0();

END_ACTION
```

#### OvlCentrovacky.st
```iecst
ACTION OvlCentrovacky:

	//Volanie funkcie SequenceControl//
	SequenceControl(SC:= SC_OvlCentrovacky);

	CASE SC_OvlCentrovacky.Step OF

		0:
			SC_OvlCentrovacky.StepName:= '0 - Nulovanie';
			Centrovacku_VYSUN:= FALSE;
			Centrovacku_ZASUN:= FALSE;

			IF SC_P1_StoperSrobovania.Step <> 0 THEN
				SC_OvlCentrovacky.ResetStep:= TRUE;
				SC_OvlCentrovacky.Step:= 1;
			END_IF

		1:
			SC_OvlCentrovacky.StepName:= '1 - Rozhodnutie o cinnosti';
			IF Centrovacku_VYSUN THEN
				SC_OvlCentrovacky.Step:= 10;
			ELSIF Centrovacku_ZASUN THEN
				SC_OvlCentrovacky.Step:= 20;
			END_IF

		10:
			SC_OvlCentrovacky.StepName:= '10 - Vysunutie centrovacky';
			SC_OvlCentrovacky.IdleTime.PT:= T#3s;
			SC_OvlCentrovacky.AlarmTime.PT:= T#6s;

			IF P1_StoperSrobovania.Automat THEN
				SC_OvlCentrovacky.AlarmTime.IN:= TRUE;
			ELSE
				SC_OvlCentrovacky.IdleTime.IN:= TRUE;
			END_IF

			IF NOT SC_OvlCentrovacky.Switch1 THEN
				P1_StoperSrobovania.OUT.Centrovanie_ZASUN:= FALSE;
                P1_StoperSrobovania.OUT.Centrovanie_VYSUN:= TRUE;
				SC_OvlCentrovacky.Switch1:= TRUE;
			END_IF

			IF P1_StoperSrobovania.IN.Centrovanie_VYSUNUTE OR SC_OvlCentrovacky.IdleTime.Q THEN
				SC_OvlCentrovacky.ResetStep:= TRUE;
				SC_OvlCentrovacky.Step:= 0;
			ELSIF SC_OvlCentrovacky.AlarmTime.Q THEN
				P1_Alarmy[111]:= TRUE;
				P1_Pracovisko.STAV.Porucha_ST2:= TRUE;
			END_IF

		20:
			SC_OvlCentrovacky.StepName:= '20 - Zasunutie centrovacky';
			SC_OvlCentrovacky.IdleTime.PT:= T#3s;
			SC_OvlCentrovacky.AlarmTime.PT:= T#6s;

			IF P1_StoperSrobovania.Automat THEN
				SC_OvlCentrovacky.AlarmTime.IN:= TRUE;
			ELSE
				SC_OvlCentrovacky.IdleTime.IN:= TRUE;
			END_IF

			IF NOT SC_OvlCentrovacky.Switch1 THEN
				P1_StoperSrobovania.OUT.Centrovanie_VYSUN:= FALSE;
                P1_StoperSrobovania.OUT.Centrovanie_ZASUN:= TRUE;
				SC_OvlCentrovacky.Switch1:= TRUE;
			END_IF

			IF P1_StoperSrobovania.IN.Centrovanie_ZASUNUTE OR SC_OvlCentrovacky.IdleTime.Q THEN
				SC_OvlCentrovacky.ResetStep:= TRUE;
				SC_OvlCentrovacky.Step:= 0;
			ELSIF SC_OvlCentrovacky.AlarmTime.Q THEN
				P1_Alarmy[112]:= TRUE;
				P1_Pracovisko.STAV.Porucha_ST2:= TRUE;
			END_IF

	END_CASE

END_ACTION
```

### Program Logical/Program/Pracovisko_1/P1_Srobovanie (IEC)
